// TIA Portal V20 export
TYPE "typeSequenceControlNodeConveyorJobInterfaceCommands"
// stored: Namespace Unit1.Em7
   STRUCT
      reqManPpUnloading { ExternalWritable := 'False'} : Bool;
      reqVisionInspection { ExternalWritable := 'False'} : Bool;
   END_STRUCT;
END_TYPE
